RoboDK station: Modify Curve Density.rdk

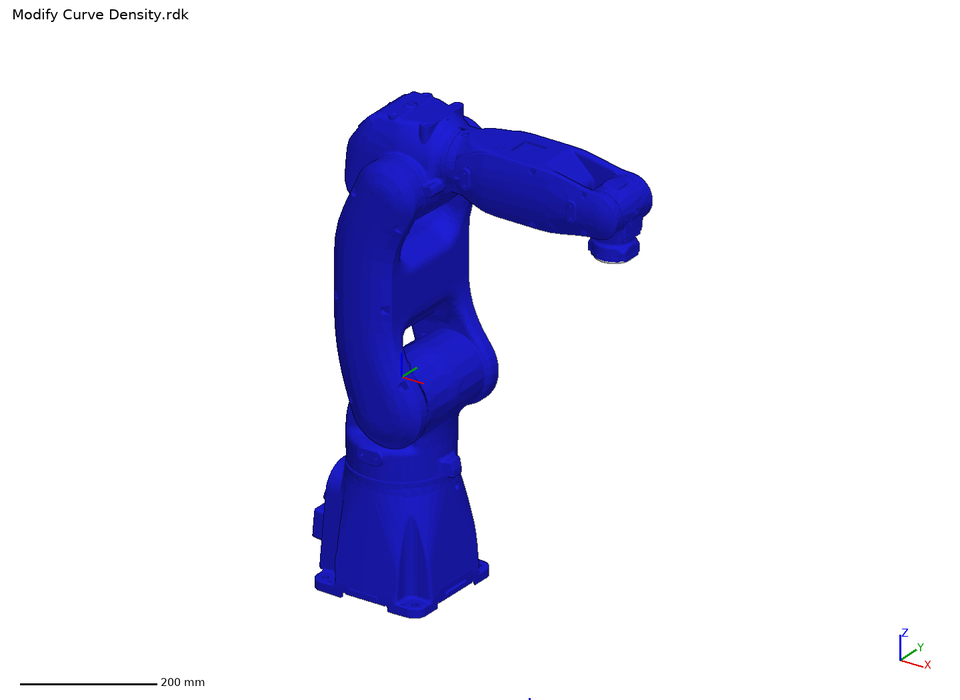
[picture v0: the station drawn from its stored meshes, robots at their saved joint values, targets as dots, program paths as lines]
Station Modify Curve Density (saved by RoboDK 5.2.1). Poses are relative to the parent item; angles as X-Y-Z fixed-axis rotations.
  - frame Motoman GP8 Base at (0, 0, 330) mm
    - robot Motoman GP8: 6 axes, payload 8 kg, reach 727 mm, repeatability 0.02 mm, weight 32 kg
        modified DH rows (alpha deg, a mm, theta deg, d mm): 0, 0, 0, 330; -90, 40, -90, 0; 0, 345, 0, 0; -90, 40, 0, 340; 90, 0, 0, 0; -90, 0, 0, 80
        base shift (0, 0, -330) mm
        joint limits [-170, -65, -113, -190, -135, -360] to [170, 150, 255, 190, 135, 360]; home [0, 0, 0, 0, 0, 0]; saved at [0, 0, 0, 0, -91.41, 0]
      - tool Tool 1, TCP at (0, 0, 100) mm
  - frame Frame 2 at (425.07, -281.48, 0) mm, rotated rx 0 ry 0 rz 90 deg
    - object Curve_Not_Enough_Points at (0, 0, 0) mm, geometry from Imported curve
  - frame Frame 3 at (635.1, -224.06, 0) mm, rotated rx 0 ry 0 rz 90 deg
    - object Curve_Too_Many_Points at (0, 0, 0) mm, geometry from LINEW=2
